// TRUE when nIn <= 0; copies nIn to nOut.
FUNCTION IsFail : BOOL
VAR_INPUT
    nIn : Result; // Result to test.
END_VAR
VAR_OUTPUT
    nOut : Result; // Copy of nIn.
END_VAR

IsFail := nIn <= 0;
nOut := nIn;

END_FUNCTION

(* stored: Version 1.1.0.1
   POU IsFail: Id {e05e24d8-50a3-4409-8484-8694994e4855}, SpecialFunc None *)
